(* IEC 61131-3 sources: iolink/src/oop, 5 files *)

(* ---- BaseIOLink.st ---- *)
USING Siemens.Simatic.S71500.DistributedIO;
NAMESPACE Simatic.Ax.iolink

    CLASS INTERNAL IOLinkBase

        VAR PROTECTED
            statDone             : Bool;                                  // Static value for output 'done'
            statBusy             : Bool;                                  // Static value for output 'busy'
            statError            : Bool;                                  // Static value for output 'error'
            statStatus           : Word := Status#STATUS_NO_CALL;         // Static value for output 'status'
            statSubfunctionStatus: DWord;                                 // Status of WRREC/RDREC or error code from IO-Link Master (%W1: IO-Link Master error, %W0: ISDU error)
			statFBErrorState     : DInt;                                  // State in the state machine of the block where the error occurred
			statFBState          : DInt := StateDevice#FB_STATE_NO_PROCESSING;  // State in the state machine of the FB
        END_VAR
        VAR PUBLIC
            Diagnostics       : LIOLink_typeDiagnostics;  // Diagnostics information of FB
        END_VAR

        METHOD PUBLIC GetStatus
            VAR_OUTPUT
                busy  : BOOL;
                error : BOOL;
                done  : BOOL;
                status : WORD;
            END_VAR

            // REGION write static values to outputs
            done := statDone;
            busy := statBusy;
            error := statError;
            status := statStatus;
            //ENO := NOT #statError;
            // END_REGION write static values to outputs
        END_METHOD

        METHOD PUBLIC Reset

            // execute reset
            statDone := FALSE;
            statBusy := FALSE;
            statError := FALSE;
            statStatus := status#STATUS_NO_CALL;

            //reset state to initial state
            statFBstate := StateDevice#FB_STATE_NO_PROCESSING;

        END_METHOD

    END_CLASS

END_NAMESPACE

(* ---- ClassDevice.st ---- *)
USING Siemens.Simatic.S71500.DistributedIO;
NAMESPACE Simatic.Ax.IOLink

    CLASS IoLinkDevice
        VAR PUBLIC
            data : LIOLink_typeRecordData;
            length : UINT;
        END_VAR
        VAR PRIVATE
			dataInternal         : LIOLink_typeRecordData;
			statDone             : Bool;                                  // Static value for output 'done'
			statBusy             : Bool;                                  // Static value for output 'busy'
			statError            : Bool;                                  // Static value for output 'error'
			statStatus           : Word := Status#STATUS_NO_CALL;         // Static value for output 'status'
			statHwID             : HW_IO;                                 // Static value for input 'hwID'
			statHwIDprevious     : HW_IO;                                 // Static value for input 'hwID' from the previous execute
			statCap              : UInt;                                  // Client Access Point (CAP) 0xB400 or 0x00E3 (227)
			statPort             : INT;                                   // Port on IO-Link master module
			statIndex            : INT;                                   // Address parameter index (IO-Link device); 0..32767: IOL-D; 65535: port functions
			statSubIndex         : INT;                                   // Address parameter subindex (IO-Link device); 0: full record; 1-255: single parameter
            statLength           : UInt;                                  // Length of data to be written to device
            statMode                : Mode;
			statPollingPeriod    : LTIME := LTIME#100MS;                       // Static value for input 'pollingPeriod'
			statTimeout          : LTIME := LTIME#20s;                         // Static value for input 'timeout'
            statRead             : LIOLink_typeReadWrite;
			statWrite            : LIOLink_typeReadWrite;
			statSubfunctionStatus: DWord;                                 // Status of WRREC/RDREC or error code from IO-Link Master (%W1: IO-Link Master error, %W0: ISDU error)
			statFBErrorState     : DInt;                                  // State in the state machine of the block where the error occurred
			statFBState          : DInt := StateDevice#FB_STATE_NO_PROCESSING;  // State in the state machine of the FB
            statBuffer           : Array[0..Lengths#RECORD_WITH_HEADER - 1] OF BYTE;
            statDiagnostics : LIOLink_typeDiagnostics;  // Diagnostics information of FB
            instRdRec            : ReadRecord;                                        // System function "read data record"
			instWrRec            : WriteRecord;                                       // System function "write data record"
			instPoll             : System.Timer.Pulse;                                // poll rate read data record
			instMonitor          : System.Timer.OnDelay;                              // request monitoring time
        END_VAR

        METHOD PUBLIC Setup
            VAR_INPUT
                hwID         : HW_IO;
                cap          : UINT;
                port         : INT;
                index        : INT;
                subindex     : INT;
                timeout      : LTIME := LTIME#20s;
                pollingPeriod: LTIME := LTIME#100ms;
            END_VAR

            statHwID := hwID;
            statcap := cap;
            statPort := port;
            statIndex := index;
            statSubIndex := subindex;
            IF timeout > LTIME#0s THEN
                statTimeout := timeout;
            END_IF;
            IF pollingPeriod > LTIME#0s THEN
                statPollingPeriod := pollingPeriod;
            END_IF;

        END_METHOD

        METHOD SetWriteCommand : BOOL
            VAR_OUTPUT
                status : WORD;
            END_VAR
            VAR_TEMP
                tempIndexCounter : INT;
            END_VAR

            IF statFBState = StateDevice#FB_STATE_NO_PROCESSING THEN
                statStatus := Status#STATUS_FIRST_CALL;
                IF length < UINT#1 OR length > TO_UINT(Lengths#RECORD) THEN
                    statStatus := Status#ERR_WRONG_LENGTH;
                    //stop execution to prohibit access out of array bounds
                    RETURN;
                END_IF;

                // REGION Build header
                // setup call header
                statWrite.header.call.port := TO_BYTE(statPort);

                // setup IOL header
                statWrite.header.iolHeader.indexLowByte := TO_BYTE(statIndex);
                statWrite.header.iolHeader.indexHighByte := TO_BYTE(SHR(TO_WORD(statIndex), UINT#8));
                statWrite.header.iolHeader.subindex := TO_BYTE(statSubindex);

                // BODY (data max. 232 Byte, Array 0..231 of Byte)
                statWrite.header.iolHeader.control := Control#CONTROL_WRITE;
                statLength := length + TO_UINT(Lengths#RECORD_HEADER); // data length header + data = IO-Link write data record
                // copy "record" to working area
                FOR tempIndexCounter := 0 TO TO_INT(length) - 1 DO
                    statWrite.data[tempIndexCounter] := data[tempIndexCounter];
                END_FOR;

                // REGION Check parameters
                // Check parameters
                IF (statPort < 0) OR (statPort > TO_INT(Limit#MAX_PORT)) THEN
                    statStatus := Status#ERR_WRONG_PORT;
                ELSIF (statIndex < 0) OR FALSE (*(statIndex > MAX_INDEX AND statIndex <> INDEX_PORT_FUNC)*) THEN //deactivate check, since it could never be valid anyway
                    statStatus := Status#ERR_WRONG_INDEX;
                ELSIF (statSubIndex < 0) OR (statSubIndex > TO_INT(Limit#MAX_SUBINDEX)) THEN
                    statStatus := Status#ERR_WRONG_SUBINDEX;

                END_IF;
                //save the hwID from the previous execute
                statHwIDprevious := statHwID;

                IF statStatus = Status#STATUS_FIRST_CALL THEN // Parameters OK
                    IF statcap <> UINT#0 THEN
                        statFBState := StateDevice#FB_STATE_PREPARE_WRITE;
                    ELSIF (statCap <> TO_UINT(Cap#CAP_STANDARD) AND statCap <> TO_UINT(Cap#CAP_LEGACY)) OR (statHwIDprevious <> statHwID) THEN // check if new device is connected => hwID changed
                        statFBState := StateDevice#FB_STATE_READ_CAP;
                    ELSE
                        statFBState := StateDevice#FB_STATE_PREPARE_WRITE;
                    END_IF;
                    //feedback, that command will be executed
                    SetWriteCommand := TRUE;
                    statBusy := TRUE;
                    statMode := Mode#WRITE;
                END_IF;
                // END_REGION
                    ;
            ELSE
                statStatus := Status#ERR_EXECUTION_ACTIVE;
            END_IF;

            //write status to output for diagnostic purposes
            status := statStatus;

        END_METHOD

        METHOD PUBLIC SetReadCommand : BOOL
            VAR_INPUT
            END_VAR
            VAR_OUTPUT
                status : WORD;
            END_VAR
            VAR_TEMP
                tempEmptyRecord : LIOLink_typeRecordData;
            END_VAR

            IF statFBState = StateDevice#FB_STATE_NO_PROCESSING THEN
                // REGION Build header
                // setup call header
                statWrite.header.call.port := TO_BYTE(statPort);

                // setup IOL header
                statWrite.header.iolHeader.indexLowByte := TO_BYTE(statIndex);
                statWrite.header.iolHeader.indexHighByte := TO_BYTE(SHR(TO_WORD(statIndex), UINT#8));
                statWrite.header.iolHeader.subindex := TO_BYTE(statSubindex);

                // BODY (data max. 232 Byte, Array 0..231 of Byte)
                // Read data record requested
                // Empty record array
                data := tempEmptyRecord;

                statWrite.header.iolHeader.control := Control#CONTROL_READ;
                statLength := TO_UINT(Lengths#RECORD_HEADER); // data length only header = IO-Link read data record
                // END_REGION

                // REGION Check parameters
                // Check parameters
                IF (statPort < 0) OR (statPort > TO_INT(Limit#MAX_PORT)) THEN
                    statStatus := Status#ERR_WRONG_PORT;
                ELSIF (statIndex < 0) OR FALSE (*(tempIndex > MAX_INDEX AND tempIndex <> INDEX_PORT_FUNC)*) THEN //deactivate check, since it could never be valid anyway
                    statStatus := Status#ERR_WRONG_INDEX;
                ELSIF (statSubindex < 0) OR (statSubindex > TO_INT(Limit#MAX_SUBINDEX)) THEN
                    statStatus := Status#ERR_WRONG_SUBINDEX;
                END_IF;
                //save the hwID from the previous execute
                statHwIDprevious := statHwID;

                IF statStatus = Status#STATUS_NO_CALL THEN // Parameters OK
                    IF statcap <> UINT#0 THEN
                        statFBState := StateDevice#FB_STATE_PREPARE_WRITE;
                    ELSIF (statCap <> TO_UINT(Cap#CAP_STANDARD) AND statCap <> TO_UINT(Cap#CAP_LEGACY)) OR (statHwIDprevious <> statHwID) THEN // check if new device is connected => hwID changed
                        statFBState := StateDevice#FB_STATE_READ_CAP;
                    ELSE
                        statFBState := StateDevice#FB_STATE_PREPARE_WRITE;
                    END_IF;
                    //feedback: request is valid and will be processed
                    SetReadCommand := TRUE;
                    statBusy := TRUE;
                    statMode := Mode#READ;
                    statStatus := Status#STATUS_SUBSEQUENT_CALL;
                END_IF;
            ELSE
                statStatus := Status#ERR_EXECUTION_ACTIVE;
            END_IF;

            //write status to output for diagnostic purposes
            status := statStatus;

        END_METHOD

        METHOD PUBLIC Execute

            VAR_TEMP
                tempIndexCounter : INT;
                temploopTest : INT;
            END_VAR

            CASE statFBState OF
                StateDevice#FB_STATE_NO_PROCESSING:
                    ; // No processing active
                    // END_REGION no processing

                    StateDevice#FB_STATE_ERROR:
                    ; //error step. Do nothing
                    //to re-enable operation, call reset()

                StateDevice#FB_STATE_READ_CAP:
                    // To find out CAP of IO-Link Master, data record with Index 16#B000 is read. If this reading was successful
                    // then CAP is 16#B400 (based on IO-Link Standard). If the reading was not successful and the status of RDREC
                    // is 16#DE80_B0xx, then CAP is 16#00E3 (227, based on Siemens Old Standard for IO-Link Masters).

                    instRdRec(record := statBuffer);

                    IF (instRdRec.BUSY = FALSE) THEN
                        IF (instRdRec.VALID = FALSE) AND (instRdRec.ERROR = FALSE) THEN
                            IF instRdRec.request = FALSE THEN
                                // call read record with Index 16#B000
                                instRdRec.request := true;
                                instRdRec.ID := statHwID;
                                instRdRec.index := TO_UINT(Cap#INDEX_CAP_IOLINK);
                                instRdRec.maxLength := UINT#0;
                                statFBState := StateDevice#FB_STATE_READ_CAP;
                            END_IF;
                        ELSIF instRdRec.VALID = TRUE THEN

                            instRdRec.request := FALSE;
                            // if status of RDREC is valid then CAP is 16#B400 (CAP_STANDARD)
                            IF instRdRec.STATUS.%B3 = ReadWriteRecordStatus#STATUS_RDREC_VALID THEN
                                statCap := TO_UINT(Cap#CAP_STANDARD);
                            END_IF;
                            statFBState := StateDevice#FB_STATE_PREPARE_WRITE;
                        ELSE
                            // if RDREC is in error state and Status is 16#DE80_B0xx then CAP is 227 (CAP_Legacy)
                            IF (instRdRec.STATUS.%B3 = BitmaskByte#BITMASK_ERR_RDREC_B3) AND (instRdRec.STATUS.%B2 = BitmaskByte#BITMASK_ERR_RDREC_B2) AND (instRdRec.STATUS.%B1 = BitmaskByte#BITMASK_ERR_RDREC_B1) THEN
                                statCap := TO_UINT(Cap#CAP_LEGACY);
                                statFBState := StateDevice#FB_STATE_PREPARE_WRITE;
                            ELSE
                                statStatus := Status#ERR_RDREC;
                                statSubfunctionStatus := instRdRec.STATUS;
                                statCap := UINT#0; //clear CAP if an error occurs
                            END_IF;
                        END_IF;
                    ELSE
                        instRdRec.request := FALSE;
                        IF instRdRec.ERROR = TRUE THEN
                            statStatus := Status#ERR_RDREC;
                            statSubfunctionStatus := instRdRec.STATUS;
                            statCap := UINT#0; //clear CAP if an error occurs
                        END_IF;
                    END_IF;

                    instRdRec(record := statBuffer);
                    // END_REGION

                StateDevice#FB_STATE_PREPARE_WRITE:

                    //read and write record system functions in SIMATIC AX are more strict
                    //it is not possible to add a struct as VAR_IN_OUT to them
                    //instead, a byte array is needed. This intermediate step converts the struct data to write into the byte array for the system function
                    SerializeBig(offset := UDINT#0, value := statWrite, buffer := statBuffer);
                    statFBState := StateDevice#FB_STATE_WRITE;

                StateDevice#FB_STATE_WRITE:
                    // To read data records, the IO-Link master modules needs to know which port is required. Therefore it is necessary
                    // to send at first a request via write data record (header, 8 byte). As response the IO-Link master module will
                    // send the required data record.

                    instWrRec(request := TRUE,
                        ID := statHwID,
                        index := statCap,
                        length := statLength,
                        record := statBuffer);

                    IF instWrRec.ERROR THEN
                        IF (instWrRec.STATUS AND BitmaskDWord#STATUS_MASK) = BitmaskDWord#STATUS_RESOURCE_BUSY THEN
                            instWrRec(request := FALSE, record := statBuffer); // Reset request
                        ELSE
                            statStatus := status#ERR_WRREC;
                            statSubfunctionStatus := instWrRec.STATUS;
                            statFBErrorState := statFBState;
                        END_IF;
                    ELSIF instWrRec.DONE = TRUE THEN
                        instWrRec(request := FALSE, record := statBuffer); // Reset request

                        //write read config into buffer
                        SerializeBig(offset := UDINT#0, value := statRead, buffer := statBuffer);
                        statFBState := StateDevice#FB_STATE_POLL;
                    END_IF;
                    // END_REGION write

                StateDevice#FB_STATE_POLL: // wait and poll for response
                    // REGION poll
                    instPoll(signal := TRUE,
                        duration := statPollingPeriod);

                    // read data record on falling edge
                    instRdRec(request := NOT instPoll.output,
                        ID := statHwID,
                        index := statCap,
                        maxLength := UINT#0, // read all data available,
                        record := statBuffer);

                    IF instRdRec.ERROR = TRUE THEN
                        IF (instRdRec.STATUS AND BitmaskDWord#STATUS_MASK) = BitmaskDWord#STATUS_RESOURCE_BUSY THEN
                            // Reset requests and try again
                            instPoll(signal := FALSE,
                            duration := statPollingPeriod);

                            instRdRec(request := FALSE,
                            record := statBuffer);
                        ELSE
                            statStatus := status#ERR_RDREC;
                            statSubfunctionStatus := instRdRec.STATUS;
                            statFBErrorState := statFBState;
                        END_IF;
                    ELSIF instRdRec.VALID THEN

                        //deserialize received data
                        DeserializeBig(offset := UDINT#0, value := statRead, buffer := statBuffer);
                        IF // check the response wether it matches the request (compare PORT, index and SUBINDEX)
                            (statWrite.header.call.port <> statRead.header.call.port)
                            OR (statWrite.header.iolHeader.indexHighByte <> statRead.header.iolHeader.indexHighByte)
                            OR (statWrite.header.iolHeader.indexLowByte <> statRead.header.iolHeader.indexLowByte)
                            OR (statWrite.header.iolHeader.subindex <> statRead.header.iolHeader.subindex)
                        THEN // read data record doesn't match the request
                            statStatus := status#ERR_INCONSISTENT_DATA;  // output status no consistent data
                        ELSIF statRead.header.iolHeader.control = Byte#16#80 THEN // check the response for IO-Link errors
                            // State 0x80 = IOL_CALL_RES PDU shows IO-Link error detect
                            statStatus := status#ERR_IO_LINK;
                            statSubfunctionStatus.%B3 := statRead.data[0]; // IO-Link master error code
                            statSubfunctionStatus.%B2 := statRead.data[1]; // IO-Link master error code
                            statSubfunctionStatus.%B1 := statRead.data[2]; // ISDU error code
                            statSubfunctionStatus.%B0 := statRead.data[3]; // ISDU additional code
                            statFBErrorState := statFBState;
                        ELSE // read data is valid
                            IF statMode = Mode#READ THEN
                                length := instRdRec.length - TO_UINT(Lengths#RECORD_HEADER);
                                // only data will be output
                                FOR tempIndexCounter := 0 TO TO_INT(instRdRec.length - TO_UINT(Lengths#RECORD_HEADER) - UINT#1) DO
                                    data[tempIndexCounter] := statRead.data[tempIndexCounter];
                                END_FOR;
                            END_IF;

                            // Reset requests
                            instRdRec(request := FALSE,
                            record := statBuffer);

                            instPoll(signal := FALSE,
                            duration := statPollingPeriod);

                            statStatus := status#STATUS_EXECUTION_FINISHED;  // request finished
                        END_IF;
                    END_IF;
                    // END_REGION poll

                ELSE // Undefined state in state machine reached
                    // REGION undefined state
                    statStatus := status#ERR_UNDEFINED_STATE;
                    // END_REGION undefined state no relevant case, ready for new request
            END_CASE;
            // END_REGION

            IF (statStatus = status#STATUS_EXECUTION_FINISHED)  THEN // Execution finished without errors
                // REGION execution finished
                statDone := TRUE;
                statBusy := FALSE;
                statError := FALSE;
                // execution aborted --> set state no processing
                statFBState := StateDevice#FB_STATE_NO_PROCESSING;
                // END_REGION execution finished

            ELSIF (statStatus.%X15 = TRUE)  THEN // Error occurred (#statStatus is 16#8000 to 16#FFFF)
                // REGION error occured
                statDone := FALSE;
                statBusy := FALSE;
                statError := TRUE;
                statCap := UINT#0; //Reset statcap, if error occurs, get cap has to be performed again
                // Write diagnostics
                statDiagnostics.status := statStatus;
                statDiagnostics.subfunctionStatus := statSubfunctionStatus;
                statDiagnostics.stateNumber := statFBErrorState;
                // Call instructions with FALSE to be ready for next job
                instWrRec(request := FALSE, record := statBuffer);

                instRdRec(request := FALSE,
                record := statBuffer);

                instPoll(signal := FALSE,
                duration := statPollingPeriod);

                statFBState := StateDevice#FB_STATE_ERROR;

            END_IF;

        END_METHOD

        METHOD PUBLIC GetStatus

            VAR_OUTPUT
                busy  : BOOL;
                error : BOOL;
                done  : BOOL;
                status : WORD;
            END_VAR

            // REGION write static values to outputs
            done := statDone;
            busy := statBusy;
            error := statError;
            status := statStatus;
            //ENO := NOT #statError;
            // END_REGION write static values to outputs
        END_METHOD

        METHOD PUBLIC Reset

            //clear internal FB calls
            instRdRec(request := FALSE,
            record := statBuffer);
            instPoll(signal := FALSE,
            duration := statPollingPeriod);

            // execute reset
            statDone := FALSE;
            statBusy := FALSE;
            statError := FALSE;
            statStatus := status#STATUS_NO_CALL;
            length := UINT#0;

            //reset state to initial state
            statFBstate := StateDevice#FB_STATE_NO_PROCESSING;

        END_METHOD

    END_CLASS

    TYPE
        Command : (READ, WRITE, DIAGNOSE);
    END_TYPE

END_NAMESPACE

(* ---- Device.st ---- *)
USING Siemens.Simatic.S71500.DistributedIO;
NAMESPACE Simatic.Ax.IOLink

    CLASS PUBLIC Device EXTENDS IOLinkBase
        VAR PUBLIC
            data : LIOLink_typeRecordData;
            length : UINT;
        END_VAR

        VAR PRIVATE
			dataInternal         : LIOLink_typeRecordData;
    		statHwID             : HW_IO;                                 // Static value for input 'hwID'
			statHwIDprevious     : HW_IO;                                 // Static value for input 'hwID' from the previous execute
			statCap              : UInt;                                  // Client Access Point (CAP) 0xB400 or 0x00E3 (227)
			statPort             : INT;                                   // Port on IO-Link master module
			statIndex            : INT;                                   // Address parameter index (IO-Link device); 0..32767: IOL-D; 65535: port functions
			statSubIndex         : INT;                                   // Address parameter subindex (IO-Link device); 0: full record; 1-255: single parameter
            statLength           : UInt;                                  // Length of data to be written to device
            statMode             : Mode;
			statPollingPeriod    : LTIME := LTIME#100MS;                       // Static value for input 'pollingPeriod'
			statTimeout          : LTIME := LTIME#20s;                         // Static value for input 'timeout'
            statRead             : LIOLink_typeReadWrite;
			statWrite            : LIOLink_typeReadWrite;
            statBuffer           : Array[0..Lengths#RECORD_WITH_HEADER - 1] OF BYTE;
            instRdRec            : ReadRecord;                                        // System function "read data record"
			instWrRec            : WriteRecord;                                       // System function "write data record"
			instPoll             : System.Timer.Pulse;                                // poll rate read data record
			instMonitor          : System.Timer.OnDelay;                              // request monitoring time
        END_VAR

        METHOD PUBLIC Setup
            VAR_INPUT
                hwID         : HW_IO;
                cap          : UINT;
                port         : INT;
                index        : INT;
                subindex     : INT;
                timeout      : LTIME := LTIME#20s;
                pollingPeriod: LTIME := LTIME#100ms;
            END_VAR

            statHwID := hwID;
            statcap := cap;
            statPort := port;
            statIndex := index;
            statSubIndex := subindex;
            IF timeout > LTIME#0s THEN
                statTimeout := timeout;
            END_IF;
            IF pollingPeriod > LTIME#0s THEN
                statPollingPeriod := pollingPeriod;
            END_IF;

        END_METHOD

        METHOD PUBLIC Read : BOOL
            VAR_OUTPUT
                status : WORD;
            END_VAR
            VAR_TEMP
                tempEmptyRecord : LIOLink_typeRecordData;
            END_VAR

            // Empty record array
            data := tempEmptyRecord;

            IF NOT THIS.ReadWriteReqInternal() THEN
                RETURN;
            END_IF;

            statWrite.header.iolHeader.control := Control#CONTROL_READ;
            statLength := TO_UINT(Lengths#RECORD_HEADER); // data length only header = IO-Link read data record
            Read := TRUE;
            statMode := Mode#READ;
            status := statStatus;

        END_METHOD

        METHOD PUBLIC Write : BOOL
            VAR_OUTPUT
                status : WORD;
            END_VAR

            IF NOT THIS.ReadWriteReqInternal() THEN
                RETURN;
            END_IF;

            //check length of write request
            IF length < UINT#1 OR length > TO_UINT(Lengths#RECORD) THEN
                statStatus := Status#ERR_WRONG_LENGTH;
                //stop execution to prohibit access out of array bounds
                RETURN;
            END_IF;

            //copy write request data to internal structure to prevent changes while executing
            statWrite.data := data;

            statWrite.header.iolHeader.control := Control#CONTROL_WRITE;
            statLength := length + TO_UINT(Lengths#RECORD_HEADER); // data length header + data = IO-Link write data record
            //set status
            Write := TRUE;
            statMode := Mode#WRITE;
            status := statStatus;

        END_METHOD

        METHOD PROTECTED ReadWriteReqInternal : BOOL

            //check internal state
            IF statFBState <> StateDevice#FB_STATE_NO_PROCESSING THEN
                statStatus := Status#ERR_EXECUTION_ACTIVE;
                RETURN;
            END_IF;

            statStatus := Status#STATUS_FIRST_CALL;

            // setup call header
            statWrite.header.call.port := TO_BYTE(statPort);

            // setup IOL header
            statWrite.header.iolHeader.indexLowByte := TO_BYTE(statIndex);
            statWrite.header.iolHeader.indexHighByte := TO_BYTE(SHR(TO_WORD(statIndex), UINT#8));
            statWrite.header.iolHeader.subindex := TO_BYTE(statSubindex);

            // Check parameters
            IF (statPort < 0) OR (statPort > TO_INT(Limit#MAX_PORT)) THEN
                statStatus := Status#ERR_WRONG_PORT;
            ELSIF (statIndex < 0) OR FALSE (*(statIndex > MAX_INDEX AND statIndex <> INDEX_PORT_FUNC)*) THEN //deactivate check, since it could never be valid anyway
                statStatus := Status#ERR_WRONG_INDEX;
            ELSIF (statSubIndex < 0) OR (statSubIndex > TO_INT(Limit#MAX_SUBINDEX)) THEN
                statStatus := Status#ERR_WRONG_SUBINDEX;
            END_IF;

            //save the hwID from the previous execute
            statHwIDprevious := statHwID;

            IF statStatus = Status#STATUS_FIRST_CALL THEN
                //found no issues, return TRUE
                ReadWriteReqInternal := TRUE;
                statBusy := TRUE;

                //check if cap needs to be read out before accessing the device
                IF statcap <> UINT#0 THEN
                    statFBState := StateDevice#FB_STATE_PREPARE_WRITE;
                ELSIF (statCap <> TO_UINT(Cap#CAP_STANDARD) AND statCap <> TO_UINT(Cap#CAP_LEGACY)) OR (statHwIDprevious <> statHwID) THEN // check if new device is connected => hwID changed
                    statFBState := StateDevice#FB_STATE_READ_CAP;
                ELSE
                    statFBState := StateDevice#FB_STATE_PREPARE_WRITE;
                END_IF;
            END_IF;

        END_METHOD

        METHOD PUBLIC Execute

            VAR_TEMP
                tempIndexCounter : INT;
                temploopTest : INT;
            END_VAR

            CASE statFBState OF
                StateDevice#FB_STATE_NO_PROCESSING:
                    ; // No processing active
                    // END_REGION no processing

                StateDevice#FB_STATE_ERROR:
                    ; //error step. Do nothing
                    //to re-enable operation, call reset()

                StateDevice#FB_STATE_READ_CAP:
                    // To find out CAP of IO-Link Master, data record with Index 16#B000 is read. If this reading was successful
                    // then CAP is 16#B400 (based on IO-Link Standard). If the reading was not successful and the status of RDREC
                    // is 16#DE80_B0xx, then CAP is 16#00E3 (227, based on Siemens Old Standard for IO-Link Masters).

                    instRdRec(record := statBuffer);

                    IF (instRdRec.BUSY = FALSE) THEN
                        IF (instRdRec.VALID = FALSE) AND (instRdRec.ERROR = FALSE) THEN
                            IF instRdRec.request = FALSE THEN
                                // call read record with Index 16#B000
                                instRdRec.request := true;
                                instRdRec.ID := statHwID;
                                instRdRec.index := TO_UINT(Cap#INDEX_CAP_IOLINK);
                                instRdRec.maxLength := UINT#0;
                                statFBState := StateDevice#FB_STATE_READ_CAP;
                            END_IF;
                        ELSIF instRdRec.VALID = TRUE THEN

                            instRdRec.request := FALSE;
                            // if status of RDREC is valid then CAP is 16#B400 (CAP_STANDARD)
                            IF instRdRec.STATUS.%B3 = ReadWriteRecordStatus#STATUS_RDREC_VALID THEN
                                statCap := TO_UINT(Cap#CAP_STANDARD);
                            END_IF;
                            statFBState := StateDevice#FB_STATE_PREPARE_WRITE;
                        ELSE
                            // if RDREC is in error state and Status is 16#DE80_B0xx then CAP is 227 (CAP_Legacy)
                            IF (instRdRec.STATUS.%B3 = BitmaskByte#BITMASK_ERR_RDREC_B3) AND (instRdRec.STATUS.%B2 = BitmaskByte#BITMASK_ERR_RDREC_B2) AND (instRdRec.STATUS.%B1 = BitmaskByte#BITMASK_ERR_RDREC_B1) THEN
                                statCap := TO_UINT(Cap#CAP_LEGACY);
                                statFBState := StateDevice#FB_STATE_PREPARE_WRITE;
                            ELSE
                                statStatus := Status#ERR_RDREC;
                                statSubfunctionStatus := instRdRec.STATUS;
                                statCap := UINT#0; //clear CAP if an error occurs
                            END_IF;
                        END_IF;
                    ELSE
                        instRdRec.request := FALSE;
                        IF instRdRec.ERROR = TRUE THEN
                            statStatus := Status#ERR_RDREC;
                            statSubfunctionStatus := instRdRec.STATUS;
                            statCap := UINT#0; //clear CAP if an error occurs
                        END_IF;
                    END_IF;

                    instRdRec(record := statBuffer);
                    // END_REGION

                StateDevice#FB_STATE_PREPARE_WRITE:

                    //read and write record system functions in SIMATIC AX are more strict
                    //it is not possible to add a struct as VAR_IN_OUT to them
                    //instead, a byte array is needed. This intermediate step converts the struct data to write into the byte array for the system function
                    SerializeBig(offset := UDINT#0, value := statWrite, buffer := statBuffer);
                    statFBState := StateDevice#FB_STATE_WRITE;

                StateDevice#FB_STATE_WRITE:
                    // To read data records, the IO-Link master modules needs to know which port is required. Therefore it is necessary
                    // to send at first a request via write data record (header, 8 byte). As response the IO-Link master module will
                    // send the required data record.

                    instWrRec(request := TRUE,
                        ID := statHwID,
                        index := statCap,
                        length := statLength,
                        record := statBuffer);

                    IF instWrRec.ERROR THEN
                        IF (instWrRec.STATUS AND BitmaskDWord#STATUS_MASK) = BitmaskDWord#STATUS_RESOURCE_BUSY THEN
                            instWrRec(request := FALSE, record := statBuffer); // Reset request
                        ELSE
                            statStatus := status#ERR_WRREC;
                            statSubfunctionStatus := instWrRec.STATUS;
                            statFBErrorState := statFBState;
                        END_IF;
                    ELSIF instWrRec.DONE = TRUE THEN
                        instWrRec(request := FALSE, record := statBuffer); // Reset request

                        //write read config into buffer
                        SerializeBig(offset := UDINT#0, value := statRead, buffer := statBuffer);
                        statFBState := StateDevice#FB_STATE_POLL;
                    END_IF;
                    // END_REGION write

                StateDevice#FB_STATE_POLL: // wait and poll for response
                    // REGION poll
                    instPoll(signal := TRUE,
                        duration := statPollingPeriod);

                    // read data record on falling edge
                    instRdRec(request := NOT instPoll.output,
                        ID := statHwID,
                        index := statCap,
                        maxLength := UINT#0, // read all data available,
                        record := statBuffer);

                    IF instRdRec.ERROR = TRUE THEN
                        IF (instRdRec.STATUS AND BitmaskDWord#STATUS_MASK) = BitmaskDWord#STATUS_RESOURCE_BUSY THEN
                            // Reset requests and try again
                            instPoll(signal := FALSE,
                            duration := statPollingPeriod);

                            instRdRec(request := FALSE,
                            record := statBuffer);
                        ELSE
                            statStatus := status#ERR_RDREC;
                            statSubfunctionStatus := instRdRec.STATUS;
                            statFBErrorState := statFBState;
                        END_IF;
                    ELSIF instRdRec.VALID THEN

                        //deserialize received data
                        DeserializeBig(offset := UDINT#0, value := statRead, buffer := statBuffer);
                        IF // check the response wether it matches the request (compare PORT, index and SUBINDEX)
                            (statWrite.header.call.port <> statRead.header.call.port)
                            OR (statWrite.header.iolHeader.indexHighByte <> statRead.header.iolHeader.indexHighByte)
                            OR (statWrite.header.iolHeader.indexLowByte <> statRead.header.iolHeader.indexLowByte)
                            OR (statWrite.header.iolHeader.subindex <> statRead.header.iolHeader.subindex)
                        THEN // read data record doesn't match the request
                            statStatus := status#ERR_INCONSISTENT_DATA;  // output status no consistent data
                        ELSIF statRead.header.iolHeader.control = Byte#16#80 THEN // check the response for IO-Link errors
                            // State 0x80 = IOL_CALL_RES PDU shows IO-Link error detect
                            statStatus := status#ERR_IO_LINK;
                            statSubfunctionStatus.%B3 := statRead.data[0]; // IO-Link master error code
                            statSubfunctionStatus.%B2 := statRead.data[1]; // IO-Link master error code
                            statSubfunctionStatus.%B1 := statRead.data[2]; // ISDU error code
                            statSubfunctionStatus.%B0 := statRead.data[3]; // ISDU additional code
                            statFBErrorState := statFBState;
                        ELSE // read data is valid
                            IF statMode = Mode#READ THEN
                                length := instRdRec.length - TO_UINT(Lengths#RECORD_HEADER);
                                // only data will be output
                                FOR tempIndexCounter := 0 TO TO_INT(instRdRec.length - TO_UINT(Lengths#RECORD_HEADER) - UINT#1) DO
                                    data[tempIndexCounter] := statRead.data[tempIndexCounter];
                                END_FOR;
                            END_IF;

                            // Reset requests
                            instRdRec(request := FALSE,
                            record := statBuffer);

                            instPoll(signal := FALSE,
                            duration := statPollingPeriod);

                            statStatus := status#STATUS_EXECUTION_FINISHED;  // request finished
                        END_IF;
                    END_IF;
                    // END_REGION poll

                ELSE // Undefined state in state machine reached
                    // REGION undefined state
                    statStatus := status#ERR_UNDEFINED_STATE;
                    // END_REGION undefined state no relevant case, ready for new request
            END_CASE;
            // END_REGION

            IF (statStatus = status#STATUS_EXECUTION_FINISHED)  THEN // Execution finished without errors
                // REGION execution finished
                statDone := TRUE;
                statBusy := FALSE;
                statError := FALSE;
                // execution aborted --> set state no processing
                statFBState := StateDevice#FB_STATE_NO_PROCESSING;
                // END_REGION execution finished

            ELSIF (statStatus.%X15 = TRUE)  THEN // Error occurred (#statStatus is 16#8000 to 16#FFFF)
                // REGION error occured
                statDone := FALSE;
                statBusy := FALSE;
                statError := TRUE;
                statCap := UINT#0; //Reset statcap, if error occurs, get cap has to be performed again
                // Write diagnostics
                Diagnostics.status := statStatus;
                Diagnostics.subfunctionStatus := statSubfunctionStatus;
                Diagnostics.stateNumber := statFBErrorState;
                // Call instructions with FALSE to be ready for next job
                instWrRec(request := FALSE, record := statBuffer);

                instRdRec(request := FALSE,
                record := statBuffer);

                instPoll(signal := FALSE,
                duration := statPollingPeriod);

                statFBState := StateDevice#FB_STATE_ERROR;

            END_IF;

        END_METHOD

        METHOD PUBLIC OVERRIDE Reset

            //clear internal FB calls
            instRdRec(request := FALSE,
            record := statBuffer);
            instPoll(signal := FALSE,
            duration := statPollingPeriod);

            length := UINT#0;

            SUPER.Reset();
        END_METHOD

    END_CLASS

END_NAMESPACE

(* ---- Diagnose.st ---- *)
USING Siemens.Simatic.S71500.DistributedIO;
NAMESPACE Simatic.Ax.IOLink

    CLASS PUBLIC Diagnose EXTENDS IOLinkBase

        VAR PUBLIC
            events     : LIOLink_typeEvents;
        END_VAR

        VAR PROTECTED
            statHwID             : HW_ANY;                                    // Static value for input 'HwID'
			statHwIDprevious     : HW_IO;                                     // Static value for input 'hwID' from the previous execute
			statEmptyDiagnostics : LIOLink_typeDiagnostics;                   // Empty diagnostics information (for initialization purposes only)
			instRdRec            : ReadRecord;                                // System function "read data record"
			instRdDiag           : ReadRecord;                                // System function "read data record"
			statDiagRecord       : Array[0..Lengths#RECORD - 1] of Byte;      // Data record of port diagnose
			statDiagRecordEco    : LIOLink_typeEvents;
			statCap              : UInt;                                      // Static value for input 'cap'
			statRead             : Array[0..Lengths#RECORD - 1] of Byte;      // Data record, Output of RDREC
			statIndexDiag        : UInt;                                      // Static value for index of data record of port diagnose
			statPortNumber       : Int := 8;                                  // Number of Ports of IO-Link-Master
			statPortEco          : UInt := UINT#1;                            // Static value for a port counter of EcoPN
        END_VAR

        VAR CONSTANT
            STATUS_MASK                             : DWord := DWORD#16#00FF_FF00;  // Mask to filter error codes
			STATUS_RESOURCE_BUSY                    : DWord := DWORD#16#0080_C200;  // Status from WRREC/RDREC: Resource is busy
            RESET_WORD                              : Word  := WORD#16#0000;        // Reset event codes0
            RESET_BYTE                              : Byte  := BYTE#16#00;          // Reset byte for statDiagRecord
            STATUS_RDREC_VALID                      : Byte  := BYTE#16#00;          // Status Code of RDREC in cased of no error occurs
            INDEX_DIAG_OTHER                        : Word  := WORD#16#00E5;        // Index for port status based on Siemens Standard (old): 229 => reads status of all ports
			INDEX_DIAG_ECO                          : Word  := WORD#16#B200;        // Index for port status based on IO-Link-Standard: 16#B20n, n:Port number => reads port status of only one port
            MASTER_PORT_STATUS_V2                   : Byte  := BYTE#16#02;          // Master port status version 2
			MASTER_PORT_STATUS_V3                   : Byte  := BYTE#16#03;          // Master port status version 3
			MASTER_PORT_STATUS_V4                   : Byte  := BYTE#16#04;          // Master port status version 4
            START_INDEX_MASTER_PORT_STATUS_V2       : Int   := 28;                  // Start index of relevant data in the case of port status version 2
			START_INDEX_MASTER_PORT_STATUS_V3       : Int   := 34;                  // Start index of relevant data in the case of port status version 3
			START_INDEX_MASTER_PORT_STATUS_V4       : Int   := 42;                  // Start index of relevant data in the case of port status version 4
			START_INDEX_MASTER_PORT_STATUS_STANDARD : Int   := 18;                  // Start index of relevant data in case of a IO-Link Standard data record for port status
        END_VAR

        METHOD PUBLIC Start : BOOL

            VAR_INPUT
                hwID   : HW_IO;  // Hardware identifier of IO-Link master module or first sub module
                cap    : Int;    // Client Access Point (CAP) 0xB400 or 0x00E3 (227)
            END_VAR
            VAR_TEMP
                tempPortNumber  : Int;    // Temporary value for port number
                tempEventNumber : Int;    // Temporary value for event number
                tempIndexDiagRec: Int;    // Temporary value for index of data record (array) of diagnose
            END_VAR

            //cancel command if the internal functionality is already active
            IF statFBState <> StateDiagnose#FB_STATE_NO_PROCESSING THEN
                RETURN;
            END_IF;

            //only allow valid hardware id
            IF hwID = WORD#0 THEN
                RETURN;
            END_IF;

            //reset diagnostic data
            statStatus := Status#STATUS_FIRST_CALL;
			statSubFunctionStatus := Status#STATUS_EXECUTION_FINISHED;
			statFBErrorState := 0;
			diagnostics := statEmptyDiagnostics;
			//save the hwID from the previous execute
			statHwIDprevious := statHwID;

			//reset static variables of Diagnose Records
			FOR tempPortNumber := 1 TO Lengths#MAX_PORTS DO
				FOR tempEventNumber := 0 TO Lengths#PORT_EVENT_CODES - 1 DO
					statDiagRecordEco.port[tempPortNumber].event[tempEventNumber].eventQualifier.instance := RESET_BYTE;
					statDiagRecordEco.port[tempPortNumber].event[tempEventNumber].eventQualifier.source := FALSE;
					statDiagRecordEco.port[tempPortNumber].event[tempEventNumber].eventQualifier.eventType := RESET_BYTE;
					statDiagRecordEco.port[tempPortNumber].event[tempEventNumber].eventQualifier.mode := RESET_BYTE;
					statDiagRecordEco.port[tempPortNumber].event[tempEventNumber].eventCode := RESET_WORD;
				END_FOR;
			END_FOR;
			FOR tempIndexDiagRec := 0 TO Lengths#RECORD - 1 DO
				statDiagRecord[tempIndexDiagRec] := RESET_BYTE;
			END_FOR;

            // Check parameters
			IF statStatus = Status#STATUS_FIRST_CALL THEN // Parameters OK
				IF cap <> 0 THEN   //check if cap is predefined, or given by the user
					statCap := TO_UINT(cap);
					statFBState := StateDiagnose#FB_STATE_READ_DIAG;
				ELSIF (statCap <> TO_UINT(Cap#CAP_STANDARD) AND statCap <> TO_UINT(Cap#CAP_LEGACY)) OR (statHwIDprevious <> hwID) THEN
					statFBState := StateDiagnose#FB_STATE_READ_CAP;
				ELSE //CAP already known
					statFBState := StateDiagnose#FB_STATE_READ_DIAG;
				END_IF;
			END_IF;
			//save current hwID
			statHwID := hwID;

            //feedback, that command will be executed
            Start := TRUE;

        END_METHOD

        METHOD PUBLIC Execute
            VAR_TEMP
                tempPortNumber  : Int;    // Temporary value for port number
                tempEventNumber : Int;    // Temporary value for event number
                tempIndexDiagRec: Int;    // Temporary value for index of data record (array) of diagnose
            END_VAR

            CASE statFBState OF // State machine of FB
                StateDiagnose#FB_STATE_NO_PROCESSING:
                    // No processing active (Note: this state must always be present and left empty)
                    ;

                StateDiagnose#FB_STATE_ERROR:
                    //error step. Do nothing
                    //to re-enable operation, call reset()
                    ;

                StateDiagnose#FB_STATE_READ_CAP:
                    // To find out CAP of IO-Link Master, data record with Index 16#B000 is read. If this reading was successful
                    // then CAP is 16#B400 (based on IO-Link Standard). If the reading was not successful and the status of RDREC
                    // is 16#DE80_B0xx, then CAP is 16#00E3 (227, based on Siemens Old Standard for IO-Link Masters).

                    instRdRec(record := statRead);

                    IF (instRdRec.BUSY = FALSE) THEN
                        IF (instRdRec.VALID = FALSE) AND (instRdRec.ERROR = FALSE) THEN
                            IF instRdRec.request = FALSE THEN
                                // call read record with Index 16#B000
                                instRdRec.request := TRUE;
                                instRdRec.ID := statHwID;
                                instRdRec.index := TO_UINT(Cap#INDEX_CAP_IOLINK);
                                instRdRec.maxLength := UINT#0;
                                statFBState := StateDiagnose#FB_STATE_READ_CAP;
                            END_IF;
                        ELSIF instRdRec.VALID = TRUE THEN
                            instRdRec.request := FALSE;
                            // if status of RDREC is valid then CAP is 16#B400 (CAP_STANDARD)
                            IF instRdRec.STATUS.%B3 = STATUS_RDREC_VALID THEN
                                statCap := TO_UINT(Cap#CAP_STANDARD);
                                statPortNumber := TO_INT(statRead[11]); //read number of ports of IO-Link-Master
                                statPortEco := UINT#1;
                                statIndexDiag := TO_UINT(INDEX_DIAG_ECO) + statPortEco; //Data Record with the status of each port: 0xB20n, n - Port number
                            END_IF;
                            statFBState := StateDiagnose#FB_STATE_READ_DIAG;
                        ELSE
                            // if RDREC is in error state and Status is 16#DE80_B0xx then CAP is 227 (CAP_Legacy)
                            IF (instRdRec.STATUS.%B3 = BitmaskByte#BITMASK_ERR_RDREC_B3) AND (instRdRec.STATUS.%B2 = BitmaskByte#BITMASK_ERR_RDREC_B2) AND (instRdRec.STATUS.%B1 = BitmaskByte#BITMASK_ERR_RDREC_B1) THEN
                                statCap := TO_UINT(Cap#CAP_LEGACY);
                                statIndexDiag := TO_UINT(INDEX_DIAG_OTHER);
                                statFBState := StateDiagnose#FB_STATE_READ_DIAG;
                            ELSE
                                statDone := FALSE;
                                statBusy := FALSE;
                                statError := TRUE;
                                statStatus := Status#ERR_RDREC;
                                statCap := UINT#0; //clear CAP if an error occurs
                                statIndexDiag := UINT#0;
                                statSubFunctionStatus := instRdRec.STATUS;
                                statFBErrorState := statFBState;
                                statFBState := StateDiagnose#FB_STATE_NO_PROCESSING;
                            END_IF;
                        END_IF;
                    ELSE
                        instRdRec.request := FALSE;
                    END_IF;

                    instRdRec(record := statRead);
                    // END_REGION

                StateDiagnose#FB_STATE_READ_DIAG:

                    // REGION read diagnosis in case of Siemens-Version //statIndex 229
                    //diagnose of all ports is read with only one call
                    IF statIndexDiag = TO_UINT(INDEX_DIAG_OTHER) THEN
                        instRdDiag(record := statDiagRecord);
                        IF (instRdDiag.BUSY = FALSE) THEN
                            IF (instRdDiag.VALID = FALSE) AND (instRdDiag.ERROR = FALSE) THEN
                                IF instRdDiag.request = FALSE THEN
                                    instRdDiag.request := TRUE;
                                    instRdDiag.ID := statHwID;
                                    instRdDiag.index := statIndexDiag;
                                    instRdDiag.maxLength := UINT#0;
                                END_IF;
                            ELSE
                                instRdDiag.request := FALSE;
                                IF instRdDiag.VALID = TRUE THEN  //Diagnose valid, statDone is true
                                    statStatus := Status#STATUS_EXECUTION_FINISHED;
                                    statFBState := StateDiagnose#FB_STATE_NO_PROCESSING;
                                    statDone := TRUE;
                                    statBusy := FALSE;
                                    statError := FALSE;
                                ELSE
                                    IF (instRdDiag.STATUS AND STATUS_MASK) <> STATUS_RESOURCE_BUSY THEN  //Error occured
                                        statDone := FALSE;
                                        statBusy := FALSE;
                                        statError := TRUE;
                                        statStatus := Status#ERR_RDREC;
                                        statCap := UINT#0;
                                        statIndexDiag := UINT#0;
                                        statSubFunctionStatus := instRdDiag.STATUS;
                                        statFBErrorState := statFBState;
                                        statFBState := StateDiagnose#FB_STATE_NO_PROCESSING;
                                    END_IF;
                                END_IF;
                            END_IF;
                        ELSE
                            instRdDiag.request := FALSE;
                        END_IF;
                        instRdDiag(record := statDiagRecord);
                    END_IF;
                    // END_REGION

                    // REGION read diagnosis in case of Standard-Version // Index 0xB20n, n - Port number
                    IF statIndexDiag = (TO_UINT(INDEX_DIAG_ECO) + statPortEco) THEN
                        //one call for each port diagnose, statPortEco starting from 1 to maximum number of ports
                        IF statPortEco < TO_UINT((statPortNumber + 1)) THEN
                            instRdDiag(record := statDiagRecord);
                            IF (instRdDiag.BUSY = FALSE) THEN
                                IF (instRdDiag.VALID = FALSE) AND (instRdDiag.ERROR = FALSE) THEN
                                    IF instRdDiag.request = FALSE THEN
                                        instRdDiag.request := TRUE;
                                        instRdDiag.ID := statHwID;
                                        instRdDiag.index := statIndexDiag;
                                        instRdDiag.maxLength := UINT#0;
                                    END_IF;
                                ELSE
                                    instRdDiag.request := FALSE;
                                    IF instRdDiag.VALID = TRUE THEN  //Diagnose of port is valid
                                        tempIndexDiagRec := START_INDEX_MASTER_PORT_STATUS_STANDARD; //starting index of data record, where events are recorded
                                        //for each port, the 5 last-events are saved in output
                                        FOR tempEventNumber := 0 TO Lengths#PORT_EVENT_CODES - 1 DO
                                            statDiagRecordEco.port[statPortEco].event[tempEventNumber].eventQualifier.instance.%X0 := statDiagRecord[tempIndexDiagRec].%X0;
                                            statDiagRecordEco.port[statPortEco].event[tempEventNumber].eventQualifier.instance.%X1 := statDiagRecord[tempIndexDiagRec].%X1;
                                            statDiagRecordEco.port[statPortEco].event[tempEventNumber].eventQualifier.instance.%X2 := statDiagRecord[tempIndexDiagRec].%X2;
                                            statDiagRecordEco.port[statPortEco].event[tempEventNumber].eventQualifier.source := statDiagRecord[tempIndexDiagRec].%X3;
                                            statDiagRecordEco.port[statPortEco].event[tempEventNumber].eventQualifier.eventType.%X0 := statDiagRecord[tempIndexDiagRec].%X4;
                                            statDiagRecordEco.port[statPortEco].event[tempEventNumber].eventQualifier.eventType.%X1 := statDiagRecord[tempIndexDiagRec].%X5;
                                            statDiagRecordEco.port[statPortEco].event[tempEventNumber].eventQualifier.mode.%X0 := statDiagRecord[tempIndexDiagRec].%X6;
                                            statDiagRecordEco.port[statPortEco].event[tempEventNumber].eventQualifier.mode.%X1 := statDiagRecord[tempIndexDiagRec].%X7;
                                            statDiagRecordEco.port[statPortEco].event[tempEventNumber].eventCode.%B1 := statDiagRecord[tempIndexDiagRec + 1];
                                            statDiagRecordEco.port[statPortEco].event[tempEventNumber].eventCode.%B0 := statDiagRecord[tempIndexDiagRec + 2];
                                            tempIndexDiagRec := tempIndexDiagRec + 3; //3-bytes for each event => 2 bytes for event code + 1 byte for event type
                                        END_FOR;
                                        statPortEco := statPortEco + UINT#1; //port number is updated => next port
                                        statIndexDiag := TO_UINT(INDEX_DIAG_ECO) + statPortEco; //change index for the next port diagnose
                                    ELSE
                                        IF (instRdDiag.STATUS AND STATUS_MASK) <> STATUS_RESOURCE_BUSY THEN  //Error occured
                                            statDone := FALSE;
                                            statBusy := FALSE;
                                            statError := TRUE;
                                            statStatus := Status#ERR_RDREC;
                                            statCap := UINT#0;
                                            statIndexDiag := UINT#0;
                                            statSubFunctionStatus := instRdDiag.STATUS;
                                            statFBErrorState := statFBState;
                                            statFBState := StateDiagnose#FB_STATE_NO_PROCESSING;
                                            statPortEco := UINT#0;
                                        END_IF;
                                    END_IF;
                                END_IF;
                            ELSE
                                instRdDiag.request := FALSE;
                            END_IF;
                            instRdDiag(record := statDiagRecord);
                        ELSE
                            //diagnose of all ports was successfully read
                            statPortEco := UINT#1;
                            statIndexDiag := TO_UINT(INDEX_DIAG_ECO) + statPortEco;
                            statStatus := Status#STATUS_EXECUTION_FINISHED;
                            statFBState := StateDiagnose#FB_STATE_NO_PROCESSING;
                            statDone := TRUE;
                            statBusy := FALSE;
                            statError := FALSE;
                        END_IF;
                    END_IF;

            ELSE // Undefined state in state machine reached
                statDone := FALSE;
                statBusy := FALSE;
                statError := TRUE;
                statStatus := Status#ERR_UNDEFINED_STATE;
            END_CASE;

            // Fill event codes in case of new received diagnosis data
            IF statDone = TRUE THEN
                IF statIndexDiag = TO_UINT(INDEX_DIAG_OTHER) THEN
                    //Diagnosis record in case of Siemens Old Standard
                    // REGION EVENTCODES_SIEMENS_VERSION
                    //The master post status record has 3 versions (1,2,3-Version). For each post status record there is a different offset, from where the diagnose data can be found.
                    //The master port status version is found in Byte 0 of each port status data record e.g. statDiagRecord[0].
                    //Therefore based on the master port status version, the start index of diagnose data is found.
                    IF statDiagRecord[0] = MASTER_PORT_STATUS_V2 THEN
                        tempIndexDiagRec := START_INDEX_MASTER_PORT_STATUS_V2;
                    ELSIF statDiagRecord[0] = MASTER_PORT_STATUS_V3 THEN
                        tempIndexDiagRec := START_INDEX_MASTER_PORT_STATUS_V3;
                    ELSIF statDiagRecord[0] = MASTER_PORT_STATUS_V4 THEN
                        tempIndexDiagRec := START_INDEX_MASTER_PORT_STATUS_V4;
                    END_IF;

                    IF (statDiagRecord[0] = MASTER_PORT_STATUS_V2) OR (statDiagRecord[0] = MASTER_PORT_STATUS_V3) OR (statDiagRecord[0] = MASTER_PORT_STATUS_V4) THEN
                        FOR tempPortNumber := 1 TO Lengths#MAX_PORTS DO
                            FOR tempEventNumber := 0 TO Lengths#PORT_EVENT_CODES - 1 DO
                                events.port[tempPortNumber].event[tempEventNumber].eventQualifier.instance.%X0 := statDiagRecord[tempIndexDiagRec].%X0;
                                events.port[tempPortNumber].event[tempEventNumber].eventQualifier.instance.%X1 := statDiagRecord[tempIndexDiagRec].%X1;
                                events.port[tempPortNumber].event[tempEventNumber].eventQualifier.instance.%X2 := statDiagRecord[tempIndexDiagRec].%X2;
                                events.port[tempPortNumber].event[tempEventNumber].eventQualifier.source := statDiagRecord[tempIndexDiagRec].%X3;
                                events.port[tempPortNumber].event[tempEventNumber].eventQualifier.eventType.%X0 := statDiagRecord[tempIndexDiagRec].%X4;
                                events.port[tempPortNumber].event[tempEventNumber].eventQualifier.eventType.%X1 := statDiagRecord[tempIndexDiagRec].%X5;
                                events.port[tempPortNumber].event[tempEventNumber].eventQualifier.mode.%X0 := statDiagRecord[tempIndexDiagRec].%X6;
                                events.port[tempPortNumber].event[tempEventNumber].eventQualifier.mode.%X1 := statDiagRecord[tempIndexDiagRec].%X7;
                                events.port[tempPortNumber].event[tempEventNumber].eventCode.%B1 := statDiagRecord[tempIndexDiagRec + 1];
                                events.port[tempPortNumber].event[tempEventNumber].eventCode.%B0 := statDiagRecord[tempIndexDiagRec + 2];
                                tempIndexDiagRec := tempIndexDiagRec + 3; //3-bits for each event, 2 bits for eventcode + 1 bit for event type
                            END_FOR;
                            tempIndexDiagRec := tempIndexDiagRec + 4; //4 bits reserved for other purposes between Port Diagnoses
                        END_FOR;
                    END_IF;
                    // END_REGION
                    //Diagnosis record in case of IO-Link-Standard
                ELSIF statIndexDiag = (TO_UINT(INDEX_DIAG_ECO) + statPortEco) THEN
                    // REGION EVENTCODES_STANDARD_VERSION
                    events := statDiagRecordEco;
                    // END_REGION
                END_IF;
            ELSIF statError = TRUE THEN  //Error occurred
                diagnostics.status := statStatus;
                diagnostics.subfunctionStatus := statSubFunctionStatus;
                diagnostics.stateNumber := statFBErrorState;
            END_IF;

        END_METHOD

        METHOD PUBLIC OVERRIDE Reset

            //clear internal FB calls
			instRdRec(request    := FALSE,
				record := statRead);

			instRdDiag(request := FALSE,
                record := statDiagRecord);

            SUPER.Reset();
        END_METHOD

    END_CLASS

END_NAMESPACE

(* ---- Master.st ---- *)
USING Siemens.Simatic.S71500.DistributedIO;
NAMESPACE Simatic.Ax.IOLink

    CLASS PUBLIC Master EXTENDS IOLinkBase
        VAR PUBLIC
            Record4Ports : REF_TO LIOLink_typeMaster4PortRecordData;
            Record8Ports : REF_TO LIOLink_typeMaster8PortRecordData;
            RecordLength : DINT;
        END_VAR

        VAR PROTECTED
            instRdRec            : ReadRecord;                                        // System function "read data record"
			instWrRec            : WriteRecord;                                       // System function "write data record"
			statRecStruct        : LIOLink_typeRecStruct;
            statHwID             : HW_IO;                                             // Static value for input 'hwID'
			statMode             : USInt;                                             // Static value for input 'mode'
			statSegment          : DInt;                                              // current segment
			statAddress          : DInt;                                              // current address
			statLen              : DInt;                                              // total length of operated data
			statBuffer           : LIOLink_typeRecordDataWithHeader;
            record : REF_TO ARRAY[*] OF BYTE;
        END_VAR

        VAR CONSTANT

			INDEX                      : USInt := USINT#120;           // Index of data record for backup/restore operations
            ERR_UNKNOWN_RECORD         : DWord := DWORD#16#DF80_B000;  // Error: Data record not known in module
        END_VAR

        METHOD PUBLIC Backup : BOOL
            VAR_INPUT
                hwID : HW_IO;
                port : masterType;
            END_VAR
            VAR_OUTPUT
                status : WORD;
            END_VAR
            VAR_TEMP
                tempIndex : INT;
                tempLimit : INT;
            END_VAR

            statHwID := hwID;
            statMode := MasterMode#BACKUP;

            IF port = masterType#INVALID THEN
                RETURN;
            END_IF;

            IF NOT THIS.CheckCommandInternal(port) THEN
                RETURN;
            END_IF;

            IF port = MasterType#FOUR_PORT THEN
                tempLimit := Lengths#MASTER_RECORD_4_PORT;
            ELSE
                tempLimit := Lengths#MASTER_RECORD_8_PORT;
            END_IF;

            // initialize data record before backup
            FOR tempIndex := 0 TO tempLimit - 1 DO
                record^[tempIndex] := BYTE#16#0;
            END_FOR;
        END_METHOD

        METHOD PUBLIC Restore : BOOL
            VAR_INPUT
                hwID : HW_IO;
                port : masterType;
            END_VAR
            VAR_OUTPUT
                status : WORD;
            END_VAR
            statHwID := hwID;
            statMode := MasterMode#RESTORE;

            IF port = masterType#INVALID THEN
                RETURN;
            END_IF;

            IF NOT THIS.CheckCommandInternal(port) THEN
                status := statStatus;
                RETURN;
            END_IF;

        END_METHOD

        METHOD PROTECTED CheckCommandInternal : BOOL
            VAR_INPUT
                masterType : MasterType;
            END_VAR

            //check internal state
            IF statFBState <> StateDevice#FB_STATE_NO_PROCESSING THEN
                statStatus := Status#ERR_EXECUTION_ACTIVE;
                RETURN;
            END_IF;

            IF statHwID = WORD#0 THEN
                statStatus := Status#ERR_HARDWARE_ID_INVALID;
                RETURN;
            END_IF;

            statStatus := Status#STATUS_FIRST_CALL;

            // Initialize internal tags
			statSegment := 0;
			statAddress := 0;
			statLen := 0;

            IF  masterType = MasterType#INVALID THEN
                statStatus := Status#ERR_ARRAY_REFERENCE;
                RETURN;
            ELSIF masterType = MasterType#FOUR_PORT THEN
                IF Record4Ports = NULL THEN
                    statStatus := Status#ERR_ARRAY_UNSUPPORTED;
                    RETURN;
                END_IF;
                record := Record4Ports;
            ELSIF masterType = MasterType#EIGHT_PORT THEN
                IF Record8Ports = NULL THEN
                    statStatus := Status#ERR_ARRAY_UNSUPPORTED;
                    RETURN;
                END_IF;
                record := Record8Ports;
            END_IF;

            //everything okay, start processing
            statFBState := StateMaster#FB_STATE_PREPARE_RESET;
            statStatus := Status#STATUS_SUBSEQUENT_CALL;

        END_METHOD

        METHOD PUBLIC Execute
            VAR_TEMP
                tempIndex : INT;
                tempLength : UINT;
            END_VAR

            CASE statFBState OF
                StateMaster#FB_STATE_NO_PROCESSING:
                    ; // No processing active
                    // END_REGION no processing

                StateMaster#FB_STATE_ERROR:
                    ; //error step. Do nothing
                    //to re-enable operation, call reset()

                StateMaster#FB_STATE_PREPARE_RESET:
                    statRecStruct.reset.ExtendedFunctionNum := FunctionType#FUNC_PUSH;
                    statRecStruct.reset.SequenceNo := SeqNoMaster#SEQ_NUM_RESET;  // reset save/restore operations

                    SerializeBig(offset := UINT#0, value := statRecStruct.reset, buffer := statBuffer);
                    statFBState := stateMaster#FB_STATE_RESET;

                StateMaster#FB_STATE_RESET:

                    instWrRec(request    := true,
                        ID     := statHwID,
                        index  := index,
                        length    := TO_UINT(Lengths#MASTER_HEADER),
                        record := statBuffer);

                    IF instWrRec.DONE = TRUE THEN
                        instWrRec(request := FALSE, record := statBuffer); // Reset request

                        IF statMode = MasterMode#BACKUP THEN
                            statFBState := stateMaster#FB_STATE_BACKUP;
                        ELSE
                            statFBState := stateMaster#FB_STATE_RESTORE;
                        END_IF;

                    ELSIF instWrRec.ERROR = TRUE AND instWrRec.STATUS = ERR_UNKNOWN_RECORD THEN
                        statStatus := Status#ERR_UNKNOWN_MODULE; // set status = unknown type of module
                        statSubfunctionStatus := instWrRec.STATUS;
                        statFBErrorState := statFBState;
                    ELSIF instWrRec.ERROR = TRUE THEN
                        statStatus := Status#ERR_WRREC;
                        statSubfunctionStatus := instWrRec.STATUS;
                        statFBErrorState := statFBState;
                    END_IF;
                    // END_REGION reset

                StateMaster#FB_STATE_BACKUP:
                    instRdRec(request    := TRUE,
                        ID     := statHwID,
                        index  := index,
                        maxLength   := TO_UINT(Lengths#MASTER_RECORD_SEGMENT_WITH_HEADER),
                        record := statBuffer);

                    // evaluation of RDREC
                    IF instRdRec.VALID = TRUE THEN
                        DeserializeBig(offset := UINT#0, value := statRecStruct.backup, buffer := statBuffer);
                        IF instRdRec.length > TO_UINT(Lengths#MASTER_HEADER) AND statRecStruct.backup.ExtendedFunctionNum = FunctionType#FUNC_PULL THEN
                            statStatus := Status#STATUS_OFFSET_BACKUP OR statRecStruct.backup.SequenceNo.%B0;  // append segment number
                            statSegment := TO_DINT(statRecStruct.backup.SequenceNo);
                            tempLength := instRdRec.length - TO_UINT(Lengths#MASTER_HEADER);

                            FOR tempIndex := 0 TO TO_INT(tempLength) - 1 DO
                                record^[tempIndex + statAddress] := statRecStruct.backup.payload[tempIndex];
                            END_FOR;

                            // add total length of data
                            statLen := statLen + tempLength;

                            // set pointer to next entry in parameter blob
                            statAddress := statAddress + tempLength;

                        ELSIF instRdRec.length = TO_UINT(Lengths#MASTER_HEADER) THEN
                            // Reset request
                            instRdRec(request    := FALSE,
                            record := statBuffer);

                            statStatus := Status#STATUS_EXECUTION_FINISHED;
                        END_IF;

                    ELSIF instRdRec.ERROR = TRUE THEN
                        statStatus            := Status#ERR_RDREC;
                        statSubfunctionStatus := instRdRec.STATUS;
                        statFBErrorState      := statFBState;
                        statLen               := instRdRec.length;
                    END_IF;
                    // END_REGION backup

                StateMaster#FB_STATE_RESTORE:
                    // load restore data segment from parameter blob (max. 234 Byte per segment)
                    IF instWrRec.BUSY = FALSE AND instWrRec.DONE = FALSE THEN // Writing hasn't started
                        statRecStruct.restore.ExtendedFunctionNum := FunctionType#FUNC_PUSH;
                        statRecStruct.restore.SequenceNo := TO_DWORD(statSegment); // sequence number
                        statStatus := Status#STATUS_OFFSET_RESTORE OR statRecStruct.restore.SequenceNo.%B0;

                        // load segment data = payload
                        FOR tempIndex := 0 TO Lengths#MASTER_RECORD_SEGMENT - 1 DO
                            statRecStruct.restore.payload[tempIndex] := record^[tempindex + statAddress];
                        END_FOR;

                        //move into buffer
                        SerializeBig(offset := UINT#0, value := statRecStruct.restore, buffer := statBuffer);

                    END_IF;

                    // write segment data
                    instWrRec(request    := TRUE,
                        ID     := statHwID,
                        index  := index,
                        length := TO_UINT(Lengths#MASTER_RECORD_SEGMENT_WITH_HEADER),
                        record := statBuffer);

                    IF instWrRec.DONE = TRUE THEN
                        statLen := statLen + Lengths#MASTER_RECORD_SEGMENT;
                        instWrRec(request := FALSE, record := statBuffer); // Reset request
                        statFBState := StateMaster#FB_STATE_VERIFY;

                    ELSIF instWrRec.ERROR = TRUE THEN
                        statStatus := Status#ERR_WRREC_RESTORE;
                        statSubfunctionStatus := instWrRec.STATUS;
                        statFBErrorState := statFBState;
                    END_IF;
                    // END_REGION restore

                StateMaster#FB_STATE_VERIFY: // Verify restore
                    // REGION verify
                    instRdRec(request    := TRUE,
                        ID     := statHwID,
                        index  := index,
                        maxLength   := TO_UINT(Lengths#MASTER_RECORD_SEGMENT_WITH_HEADER),
                        record := statBuffer);

                        DeserializeBig(offset := UINT#0, value := statRecStruct.backup, buffer := statBuffer);

                    IF instRdRec.VALID = TRUE AND statRecStruct.backup.ExtendedFunctionNum = FunctionType#FUNC_PULL THEN
                        IF statRecStruct.backup.SequenceNo = SeqNoMaster#SEQ_NUM_RESTORE_ONGOING
                            OR statRecStruct.backup.SequenceNo = SeqNoMaster#SEQ_NUM_ACTIVATION_ONGOING
                        THEN
                            statSegment := statSegment + 1;
                            statAddress := statAddress + Lengths#MASTER_RECORD_SEGMENT;

                            // Reset request
                            instRdRec(request    := FALSE,
                            record := statBuffer);

                            statFBState := StateMaster#FB_STATE_RESTORE;
                            ELSIF statRecStruct.backup.SequenceNo = SeqNoMaster#SEQ_NUM_ACTIVATION_DONE THEN //
                            // Reset request
                            instRdRec(request    := FALSE,
                            record := statBuffer);

                            statStatus := Status#STATUS_EXECUTION_FINISHED;
                        ELSIF statRecStruct.backup.SequenceNo = SeqNoMaster#SEQ_NUM_CRC_FAILED
                            OR statRecStruct.backup.SequenceNo = SeqNoMaster#SEQ_NUM_BLOB_INVALID
                            OR statRecStruct.backup.SequenceNo = SeqNoMaster#SEQ_NUM_WRONG_SEQUENCE
                            OR statRecStruct.backup.SequenceNo = SeqNoMaster#SEQ_NUM_WRONG_SIZE
                        THEN
                            statStatus := Status#ERR_SEQ_NUMBER;
                            statSubfunctionStatus := statRecStruct.backup.SequenceNo;
                            statFBErrorState := statFBState;
                        END_IF;
                    ELSIF instRdRec.ERROR = TRUE THEN
                        statStatus := Status#ERR_RDREC_VERIFY;
                        statSubfunctionStatus := instRdRec.STATUS;
                        statFBErrorState := statFBState;
                    END_IF;
                    // END_REGION verify

                ELSE // Undefined state in state machine reached
                    // REGION undefined state
                    statStatus := Status#ERR_UNDEFINED_STATE;
                    // END_REGION undefined state no relevant case, ready for new request
            END_CASE;

            // Write outputs
		IF (statStatus = Status#STATUS_EXECUTION_FINISHED) AND (statDone = FALSE) THEN // Execution finished without errors
			// REGION execution finished
			statDone  := TRUE;
			statBusy  := FALSE;
			statError := FALSE;
			RecordLength := statLen;
			// execution aborted --> set state no processing
			statFBState := StateMaster#FB_STATE_NO_PROCESSING;
			// END_REGION execution finished

		ELSIF (statStatus.%X15 = TRUE) AND (statError = FALSE) THEN // Error occurred (#statStatus is 16#8000 to 16#FFFF)
			// REGION error occured
			statDone  := FALSE;
			statBusy  := FALSE;
			statError := TRUE;
			// Write diagnostics
			Diagnostics.status            := statStatus;
			Diagnostics.subfunctionStatus := statSubfunctionStatus;
			Diagnostics.stateNumber       := statFBErrorState;
			// Call instructions with FALSE to be ready for next job
			instRdRec(request    := FALSE,
				record := statBuffer);

			instWrRec(request := FALSE,
                record := statBuffer);
			// execution aborted --> set state no processing
			statFBState := StateMaster#FB_STATE_ERROR;
            RecordLength := 0;

		END_IF;

        END_METHOD

        METHOD PUBLIC OVERRIDE Reset

            //clear internal FB calls
			instRdRec(request    := FALSE,
				record := statBuffer);

			instWrRec(request := FALSE,
                record := statBuffer);

            RecordLength := 0;

            SUPER.Reset();
        END_METHOD

    END_CLASS

END_NAMESPACE
